(* CoDeSys 2.3.9.22 project: svetofor_iz_darkneta.pro *)
(* Libraries: Standard.LIB 4.10.05 11:14:46 *)

(* Global variable list: Global_Variables *)
VAR_GLOBAL
	in:BOOL;
	l1_green:BOOL;
	l1_yellow:BOOL;
	l1_red:BOOL;
	l2_green:BOOL;
	l2_yellow:BOOL;
	l2_red:BOOL;
END_VAR

(* POU PLC_PRG, CFC *)
PROGRAM PLC_PRG
VAR
	light1:TRAFFICSIGNAL;
	light2:TRAFFICSIGNAL;

END_VAR
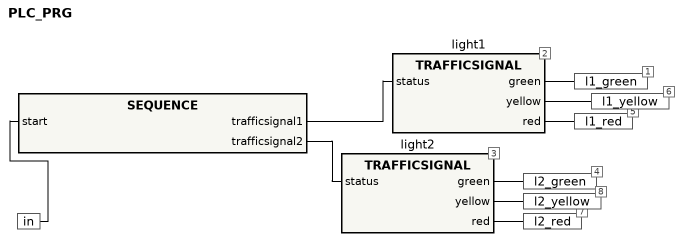
_CFC_ (* Continuous Function Chart, elements in execution order *)
#0 SEQUENCE(start: in)
#1 l1_green <= #2.green
#2 light1:TRAFFICSIGNAL(status: #0.trafficsignal1)
#3 light2:TRAFFICSIGNAL(status: #0.trafficsignal2)
#4 l2_green <= #3.green
#5 l1_red <= #2.red
#6 l1_yellow <= #2.yellow
#7 l2_red <= #3.red
#8 l2_yellow <= #3.yellow
_END_CFC_
(* the same logic as Structured Text *)
SEQUENCE(start := in);
l1_green := light1.green;
light1(status := SEQUENCE.trafficsignal1);
light2(status := SEQUENCE.trafficsignal2);
l2_green := light2.green;
l1_red := light1.red;
l1_yellow := light1.yellow;
l2_red := light2.red;
l2_yellow := light2.yellow;
END_PROGRAM

(* POU TRAFFICSIGNAL, FBD *)
FUNCTION_BLOCK TRAFFICSIGNAL
VAR_INPUT
	status:INT;
END_VAR
VAR_OUTPUT
	green:BOOL;
	yellow:BOOL;
	red:BOOL;
END_VAR
VAR
	off: BOOL;
END_VAR
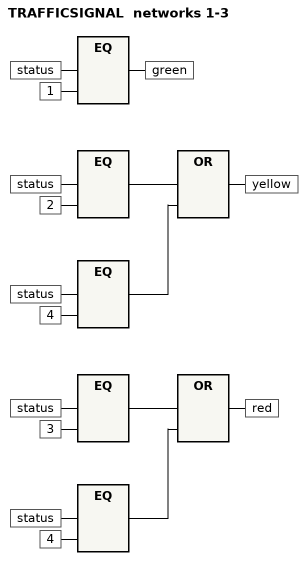
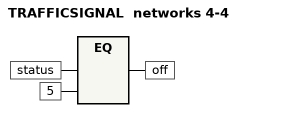
_FBD_ (* Function Block Diagram *)
NETWORK 1
	EQ(status, 1) => green
NETWORK 2
	OR(EQ(status, 2), EQ(status, 4)) => yellow
NETWORK 3
	OR(EQ(status, 3), EQ(status, 4)) => red
NETWORK 4
	EQ(status, 5) => off
_END_FBD_
(* the same logic as Structured Text *)
(* Network 1 *)
green := status = 1;
(* Network 2 *)
yellow := (status = 2) OR (status = 4);
(* Network 3 *)
red := (status = 3) OR (status = 4);
(* Network 4 *)
off := status = 5;
END_FUNCTION_BLOCK

(* POU SEQUENCE, SFC *)
PROGRAM SEQUENCE
VAR_INPUT
	start:BOOL;
END_VAR
VAR_OUTPUT
	trafficsignal1:INT;
	trafficsignal2:INT;
END_VAR
VAR
	counter:INT;
	delay:WAIT;
END_VAR
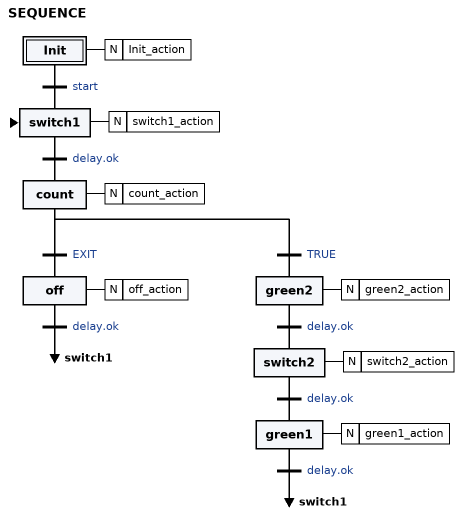
INITIAL_STEP Init:
	Init_action(N);
END_STEP
TRANSITION FROM Init TO switch1 := start;
END_TRANSITION
STEP switch1:
	switch1_action(N);
END_STEP
TRANSITION FROM switch1 TO count := delay.ok;
END_TRANSITION
STEP count:
	count_action(N);
END_STEP
TRANSITION FROM count TO off := EXIT;
END_TRANSITION
TRANSITION FROM count TO green2 := TRUE;
END_TRANSITION
STEP off:
	off_action(N);
END_STEP
TRANSITION FROM off TO switch1 := delay.ok;
END_TRANSITION
STEP green2:
	green2_action(N);
END_STEP
TRANSITION FROM green2 TO switch2 := delay.ok;
END_TRANSITION
STEP switch2:
	switch2_action(N);
END_STEP
TRANSITION FROM switch2 TO green1 := delay.ok;
END_TRANSITION
STEP green1:
	green1_action(N);
END_STEP
TRANSITION FROM green1 TO switch1 := delay.ok;
END_TRANSITION

ACTION Init_action:
	LD		1
	ST		trafficsignal1
	LD		3
	ST		trafficsignal2
END_ACTION

ACTION switch1_action:
	LD		2
	ST		trafficsignal1
	LD		4
	ST		trafficsignal2
	CAL		delay(time_in:=t#2s)
END_ACTION

ACTION count_action:
	LD		counter
	ADD		1
	ST		counter
END_ACTION

ACTION off_action:
	LD		5
	ST		trafficsignal1
	LD		5
	ST		trafficsignal2
	LD		0
	ST		counter
	CAL		delay(time_in:=t#10s)
END_ACTION

ACTION green2_action:
	LD		3
	ST		trafficsignal1
	LD		1
	ST		trafficsignal2
	CAL		delay(time_in:=t#5s)
END_ACTION

ACTION switch2_action:
	LD		4
	ST		trafficsignal1
	LD		2
	ST		trafficsignal2
	CAL		delay(time_in:=t#2s)
END_ACTION

ACTION green1_action:
	LD		1
	ST		trafficsignal1
	LD		3
	ST		trafficsignal2
	CAL		delay(time_in:=t#5s)
END_ACTION

TRANSITION EXIT:
	LD		counter
	GT		7
END_TRANSITION
END_PROGRAM

(* POU WAIT, IL *)
FUNCTION_BLOCK WAIT
VAR_INPUT
	time_in:TIME;
END_VAR
VAR_OUTPUT
	ok:BOOL:=FALSE;
END_VAR
VAR
	zab:TP;
END_VAR
	LD		zab.Q
	JMPC	mark

	CAL		zab(in:=FALSE)
	LD		time_in
	ST		zab.PT
	CAL		zab(in:=TRUE)
	JMP		end

mark:
	CAL		zab
end:
	LDN		zab.Q
	ST		ok
END_FUNCTION_BLOCK
